// TIA Portal V15.1 export
// export: Created 2020-06-12T07:35:41.5068359Z, ExportSetting None, DisplayName Totally Integrated Automation Portal, DisplayVersion V15.1, DisplayName TIA Portal Openness, DisplayVersion V15.1, DisplayName STEP 7 Professional, DisplayVersion V15.1, DisplayName STEP 7 Safety, DisplayVersion V15.1, DisplayName WinCC Advanced, DisplayVersion V15.1
FUNCTION "ES1_EMER" : Void   // FC202, FBD
TITLE = General emergency voltages (for Supply motors and valves)
{ S7_Optimized_Access := 'FALSE' }
// stored: AutoNumber false, SetENOAutomatically False
   VAR_TEMP
      _mains_ok : Bool;
   END_VAR
BEGIN

REGION Network 1: Emergency circuit is ok
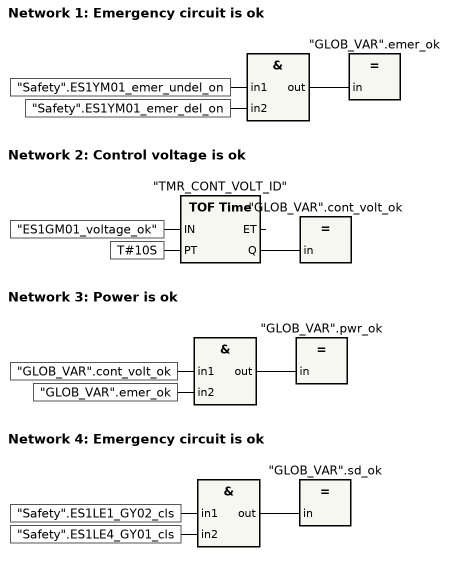
   "GLOB_VAR".emer_ok := "Safety".ES1YM01_emer_undel_on AND "Safety".ES1YM01_emer_del_on;
END_REGION

REGION Network 2: Control voltage is ok
   // "ES1GM01_main_pwr_on"
   "TMR_CONT_VOLT_ID".TOF(IN := "ES1GM01_voltage_ok", PT := T#10S);
   "GLOB_VAR".cont_volt_ok := "TMR_CONT_VOLT_ID".Q;
END_REGION

REGION Network 3: Power is ok
   // "ES1GM01_main_pwr_on"
   "GLOB_VAR".pwr_ok := "GLOB_VAR".cont_volt_ok AND "GLOB_VAR".emer_ok;
END_REGION

REGION Network 4: Emergency circuit is ok
   "GLOB_VAR".sd_ok := "Safety".ES1LE1_GY02_cls AND "Safety".ES1LE4_GY01_cls;
END_REGION
END_FUNCTION
